// TIA Portal V18 export
// export: Created 2025-12-01T12:38:33.634491Z, ExportSetting None, DisplayName Totally Integrated Automation Portal, DisplayVersion V18 Update 5, DisplayName TIA Portal Openness, DisplayVersion V18 Update 5, DisplayName TIA Portal Teamcenter Gateway, DisplayVersion V18, DisplayName TIA Portal Version Control Interface, DisplayVersion V18, DisplayName STEP 7 Professional, DisplayVersion V18 Update 5, DisplayName STEP 7 Safety, DisplayVersion V18, DisplayName WinCC Professional, DisplayVersion V18 Update 5
FUNCTION "ST10Cyl_interface31-40" : Void   // FC1023, LAD
{ S7_Optimized_Access := 'FALSE' }
// stored: AutoNumber false, SetENOAutomatically false
   VAR_INPUT
      AlwaysON : Bool;
      E_stop : Bool;
   END_VAR
   VAR_TEMP
      tTest : Bool;
   END_VAR
BEGIN

REGION Network 1 (SCL): Cylinder 31-40 IO Interface (SCL)

   //Cylinder31 IO  J-magnetLiftingLiftingCylinder
   //Input
   "ST10Cylinder".Cy[31].In.WorkPositionSensor := "iJ-magnetLiftingLiftingCylinderInWP";
   "ST10Cylinder".Cy[31].In.HomePositionSensor := "iJ-magnetLiftingLiftingCylinderInHP";
   //Output
   "oJ-magnetLiftingLiftingCylinderToWP" := "ST10Cylinder".Cy[31].Out.GoWorkPosition;
   "oJ-magnetLiftingLiftingCylinderToHP" := "ST10Cylinder".Cy[31].Out.GoHomePosition;

   //Cylinder32 IO  J-magnetLiftingPalletLocationCylinder
   //Input
   "ST10Cylinder".Cy[32].In.WorkPositionSensor := "iJ-magnetLiftingPalletLocationCylinderInWP";
   "ST10Cylinder".Cy[32].In.HomePositionSensor := "iJ-magnetLiftingPalletLocationCylinderInHP";
   //Output
   "oJ-magnetLiftingPalletLocationCylinderToWP" := "ST10Cylinder".Cy[32].Out.GoWorkPosition;
   "oJ-magnetLiftingPalletLocationCylinderToHP" := "ST10Cylinder".Cy[32].Out.GoHomePosition;

   //Cylinder33 IO  J-magnetLoadingStopperCylinder1
   //Input
   "ST10Cylinder".Cy[33].In.WorkPositionSensor := "oJ-magnetLoadingStopperCylinder1_ToWP";
   "ST10Cylinder".Cy[33].In.HomePositionSensor := "oJ-magnetLoadingStopperCylinder1_ToHP";
   //Output
   "oJ-magnetLoadingStopperCylinder1_ToWP" := "ST10Cylinder".Cy[33].Out.GoWorkPosition;
   "oJ-magnetLoadingStopperCylinder1_ToHP" := "ST10Cylinder".Cy[33].Out.GoHomePosition;

   //Cylinder34 IO  J-magnetLoadingStopperCylinder2
   //Input
   "ST10Cylinder".Cy[34].In.WorkPositionSensor := "oJ-magnetLoadingStopperCylinder2_ToWP";
   "ST10Cylinder".Cy[34].In.HomePositionSensor := "oJ-magnetLoadingStopperCylinder2_ToHP";
   //Output
   "oJ-magnetLoadingStopperCylinder2_ToWP" := "ST10Cylinder".Cy[34].Out.GoWorkPosition;
   "oJ-magnetLoadingStopperCylinder2_ToHP" := "ST10Cylinder".Cy[34].Out.GoHomePosition;

   //Cylinder35 IO  J-magnetLoadingStopperCylinder3
   //Input
   "ST10Cylinder".Cy[35].In.WorkPositionSensor := "oJ-magnetLoadingStopperCylinder3_ToWP";
   "ST10Cylinder".Cy[35].In.HomePositionSensor := "oJ-magnetLoadingStopperCylinder3_ToHP";
   //Output
   "oJ-magnetLoadingStopperCylinder3_ToWP" := "ST10Cylinder".Cy[35].Out.GoWorkPosition;
   "oJ-magnetLoadingStopperCylinder3_ToHP" := "ST10Cylinder".Cy[35].Out.GoHomePosition;

   //Cylinder36 J-magnetLoadingStopperCylinder4
   //Input
   "ST10Cylinder".Cy[36].In.WorkPositionSensor := "oJ-magnetLoadingStopperCylinder4_ToWP";
   "ST10Cylinder".Cy[36].In.HomePositionSensor := "oJ-magnetLoadingStopperCylinder4_ToHP";
   //Output
   "oJ-magnetLoadingStopperCylinder4_ToWP" := "ST10Cylinder".Cy[36].Out.GoWorkPosition;
   "oJ-magnetLoadingStopperCylinder4_ToHP" := "ST10Cylinder".Cy[36].Out.GoHomePosition;

   //Cylinder37 J-magnetTakeStopperCylinder1
   //Input
   "ST10Cylinder".Cy[37].In.WorkPositionSensor := "oJ-magnetTakeStopperCylinder1_ToWP";
   "ST10Cylinder".Cy[37].In.HomePositionSensor := "oJ-magnetTakeStopperCylinder1_ToHP";
   //Output
   "oJ-magnetTakeStopperCylinder1_ToWP" := "ST10Cylinder".Cy[37].Out.GoWorkPosition;
   "oJ-magnetTakeStopperCylinder1_ToHP" := "ST10Cylinder".Cy[37].Out.GoHomePosition;

   //Cylinder38 J-magnetTakeStopperCylinder2
   //Input
   "ST10Cylinder".Cy[38].In.WorkPositionSensor := "oJ-magnetTakeStopperCylinder2_ToWP";
   "ST10Cylinder".Cy[38].In.HomePositionSensor := "oJ-magnetTakeStopperCylinder2_ToHP";
   //Output
   "oJ-magnetTakeStopperCylinder2_ToWP" := "ST10Cylinder".Cy[38].Out.GoWorkPosition;
   "oJ-magnetTakeStopperCylinder2_ToHP" := "ST10Cylinder".Cy[38].Out.GoHomePosition;

   //Cylinder39 J-magnetTakeStopperCylinder3
   //Input
   "ST10Cylinder".Cy[39].In.WorkPositionSensor := "oJ-magnetTakeStopperCylinder3_ToWP";
   "ST10Cylinder".Cy[39].In.HomePositionSensor := "oJ-magnetTakeStopperCylinder3_ToHP";
   //Output
   "oJ-magnetTakeStopperCylinder3_ToWP" := "ST10Cylinder".Cy[39].Out.GoWorkPosition;
   "oJ-magnetTakeStopperCylinder3_ToHP" := "ST10Cylinder".Cy[39].Out.GoHomePosition;

   (*
   //Cylinder40 J-magnetLoadingStopperCylinder4_2
   // //Input
   "ST10Cylinder".Cy[40].In.WorkPositionSensor := "oJ-magnetLoadingStopperCylinder4_2";
   "ST10Cylinder".Cy[40].In.HomePositionSensor := NOT "oJ-magnetLoadingStopperCylinder4_2";
   // //Output
   "oJ-magnetLoadingStopperCylinder4_2" := "ST10Cylinder".Cy[40].Out.GoWorkPosition;
   "Feeding washer  lift Cylinder ToHP" := "ST10Cylinder".Cy[40].Out.GoHomePosition;
   *)
END_REGION

REGION Network 2: CY31 interface J-magnetLiftingLiftingCylinder
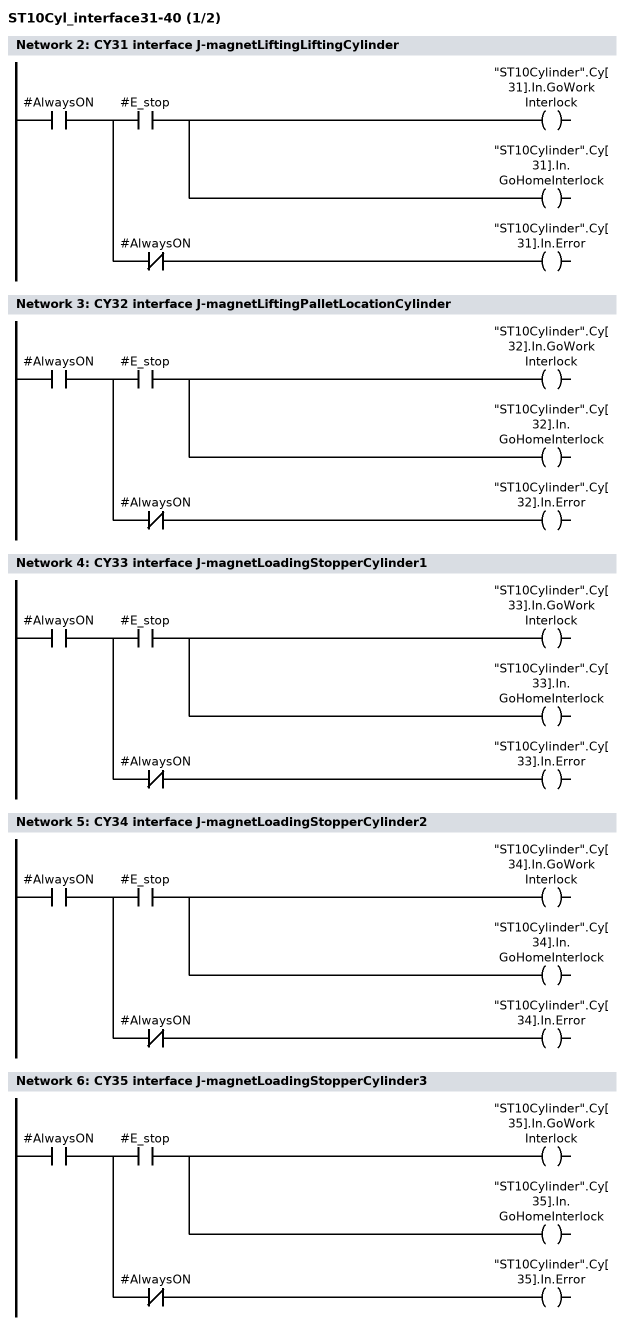
   RUNG wire#powerrail
      Contact( #AlwaysON )
      wire#w1
      Contact( #E_stop )
      wire#w2
      Coil( "ST10Cylinder".Cy[31].In.GoWorkInterlock )
   END_RUNG
   RUNG wire#w2
      Coil( "ST10Cylinder".Cy[31].In.GoHomeInterlock )
   END_RUNG
   RUNG wire#w1
      I_Contact( #AlwaysON )
      Coil( "ST10Cylinder".Cy[31].In.Error )
   END_RUNG
   // the same network as SCL:
   "ST10Cylinder".Cy[31].In.GoWorkInterlock := #AlwaysON AND #E_stop;
   "ST10Cylinder".Cy[31].In.GoHomeInterlock := #AlwaysON AND #E_stop;
   "ST10Cylinder".Cy[31].In.Error := #AlwaysON AND NOT #AlwaysON;
END_REGION

REGION Network 3: CY32 interface J-magnetLiftingPalletLocationCylinder
   RUNG wire#powerrail
      Contact( #AlwaysON )
      wire#w1
      Contact( #E_stop )
      wire#w2
      Coil( "ST10Cylinder".Cy[32].In.GoWorkInterlock )
   END_RUNG
   RUNG wire#w2
      Coil( "ST10Cylinder".Cy[32].In.GoHomeInterlock )
   END_RUNG
   RUNG wire#w1
      I_Contact( #AlwaysON )
      Coil( "ST10Cylinder".Cy[32].In.Error )
   END_RUNG
   // the same network as SCL:
   "ST10Cylinder".Cy[32].In.GoWorkInterlock := #AlwaysON AND #E_stop;
   "ST10Cylinder".Cy[32].In.GoHomeInterlock := #AlwaysON AND #E_stop;
   "ST10Cylinder".Cy[32].In.Error := #AlwaysON AND NOT #AlwaysON;
END_REGION

REGION Network 4: CY33 interface J-magnetLoadingStopperCylinder1
   RUNG wire#powerrail
      Contact( #AlwaysON )
      wire#w1
      Contact( #E_stop )
      wire#w2
      Coil( "ST10Cylinder".Cy[33].In.GoWorkInterlock )
   END_RUNG
   RUNG wire#w2
      Coil( "ST10Cylinder".Cy[33].In.GoHomeInterlock )
   END_RUNG
   RUNG wire#w1
      I_Contact( #AlwaysON )
      Coil( "ST10Cylinder".Cy[33].In.Error )
   END_RUNG
   // the same network as SCL:
   "ST10Cylinder".Cy[33].In.GoWorkInterlock := #AlwaysON AND #E_stop;
   "ST10Cylinder".Cy[33].In.GoHomeInterlock := #AlwaysON AND #E_stop;
   "ST10Cylinder".Cy[33].In.Error := #AlwaysON AND NOT #AlwaysON;
END_REGION

REGION Network 5: CY34 interface J-magnetLoadingStopperCylinder2
   RUNG wire#powerrail
      Contact( #AlwaysON )
      wire#w1
      Contact( #E_stop )
      wire#w2
      Coil( "ST10Cylinder".Cy[34].In.GoWorkInterlock )
   END_RUNG
   RUNG wire#w2
      Coil( "ST10Cylinder".Cy[34].In.GoHomeInterlock )
   END_RUNG
   RUNG wire#w1
      I_Contact( #AlwaysON )
      Coil( "ST10Cylinder".Cy[34].In.Error )
   END_RUNG
   // the same network as SCL:
   "ST10Cylinder".Cy[34].In.GoWorkInterlock := #AlwaysON AND #E_stop;
   "ST10Cylinder".Cy[34].In.GoHomeInterlock := #AlwaysON AND #E_stop;
   "ST10Cylinder".Cy[34].In.Error := #AlwaysON AND NOT #AlwaysON;
END_REGION

REGION Network 6: CY35 interface J-magnetLoadingStopperCylinder3
   RUNG wire#powerrail
      Contact( #AlwaysON )
      wire#w1
      Contact( #E_stop )
      wire#w2
      Coil( "ST10Cylinder".Cy[35].In.GoWorkInterlock )
   END_RUNG
   RUNG wire#w2
      Coil( "ST10Cylinder".Cy[35].In.GoHomeInterlock )
   END_RUNG
   RUNG wire#w1
      I_Contact( #AlwaysON )
      Coil( "ST10Cylinder".Cy[35].In.Error )
   END_RUNG
   // the same network as SCL:
   "ST10Cylinder".Cy[35].In.GoWorkInterlock := #AlwaysON AND #E_stop;
   "ST10Cylinder".Cy[35].In.GoHomeInterlock := #AlwaysON AND #E_stop;
   "ST10Cylinder".Cy[35].In.Error := #AlwaysON AND NOT #AlwaysON;
END_REGION

REGION Network 7: CY36 interface J-magnetLoadingStopperCylinder4
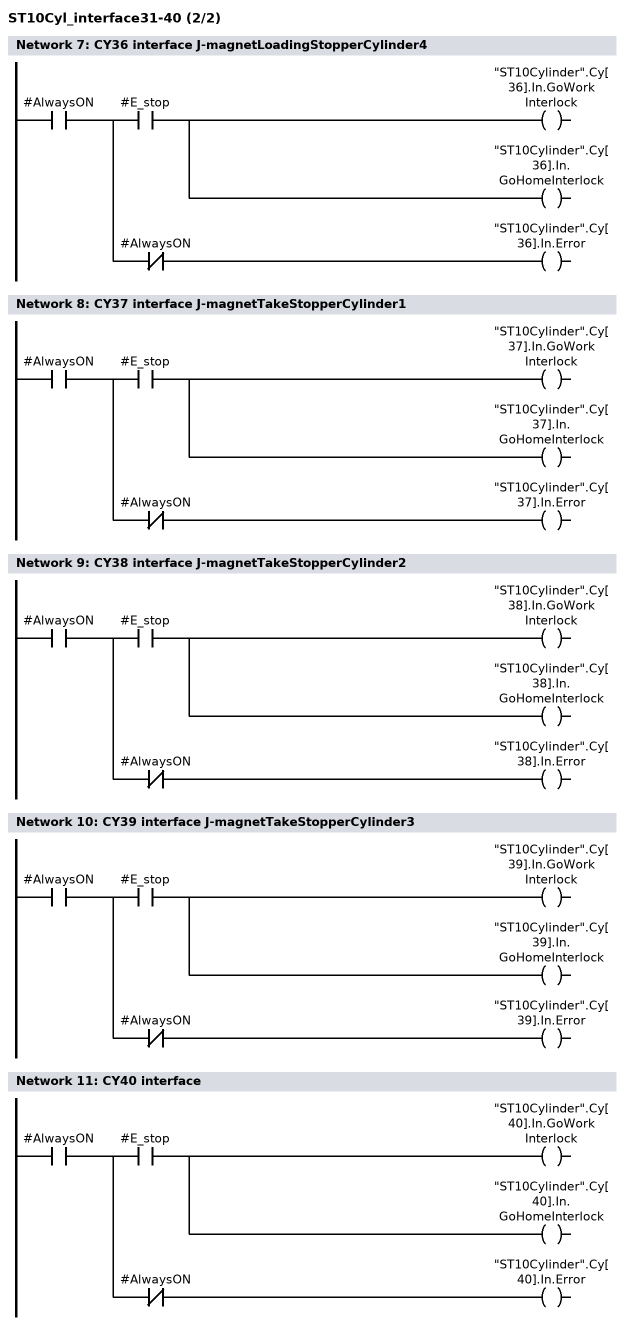
   RUNG wire#powerrail
      Contact( #AlwaysON )
      wire#w1
      Contact( #E_stop )
      wire#w2
      Coil( "ST10Cylinder".Cy[36].In.GoWorkInterlock )
   END_RUNG
   RUNG wire#w2
      Coil( "ST10Cylinder".Cy[36].In.GoHomeInterlock )
   END_RUNG
   RUNG wire#w1
      I_Contact( #AlwaysON )
      Coil( "ST10Cylinder".Cy[36].In.Error )
   END_RUNG
   // the same network as SCL:
   "ST10Cylinder".Cy[36].In.GoWorkInterlock := #AlwaysON AND #E_stop;
   "ST10Cylinder".Cy[36].In.GoHomeInterlock := #AlwaysON AND #E_stop;
   "ST10Cylinder".Cy[36].In.Error := #AlwaysON AND NOT #AlwaysON;
END_REGION

REGION Network 8: CY37 interface J-magnetTakeStopperCylinder1
   RUNG wire#powerrail
      Contact( #AlwaysON )
      wire#w1
      Contact( #E_stop )
      wire#w2
      Coil( "ST10Cylinder".Cy[37].In.GoWorkInterlock )
   END_RUNG
   RUNG wire#w2
      Coil( "ST10Cylinder".Cy[37].In.GoHomeInterlock )
   END_RUNG
   RUNG wire#w1
      I_Contact( #AlwaysON )
      Coil( "ST10Cylinder".Cy[37].In.Error )
   END_RUNG
   // the same network as SCL:
   "ST10Cylinder".Cy[37].In.GoWorkInterlock := #AlwaysON AND #E_stop;
   "ST10Cylinder".Cy[37].In.GoHomeInterlock := #AlwaysON AND #E_stop;
   "ST10Cylinder".Cy[37].In.Error := #AlwaysON AND NOT #AlwaysON;
END_REGION

REGION Network 9: CY38 interface J-magnetTakeStopperCylinder2
   RUNG wire#powerrail
      Contact( #AlwaysON )
      wire#w1
      Contact( #E_stop )
      wire#w2
      Coil( "ST10Cylinder".Cy[38].In.GoWorkInterlock )
   END_RUNG
   RUNG wire#w2
      Coil( "ST10Cylinder".Cy[38].In.GoHomeInterlock )
   END_RUNG
   RUNG wire#w1
      I_Contact( #AlwaysON )
      Coil( "ST10Cylinder".Cy[38].In.Error )
   END_RUNG
   // the same network as SCL:
   "ST10Cylinder".Cy[38].In.GoWorkInterlock := #AlwaysON AND #E_stop;
   "ST10Cylinder".Cy[38].In.GoHomeInterlock := #AlwaysON AND #E_stop;
   "ST10Cylinder".Cy[38].In.Error := #AlwaysON AND NOT #AlwaysON;
END_REGION

REGION Network 10: CY39 interface J-magnetTakeStopperCylinder3
   RUNG wire#powerrail
      Contact( #AlwaysON )
      wire#w1
      Contact( #E_stop )
      wire#w2
      Coil( "ST10Cylinder".Cy[39].In.GoWorkInterlock )
   END_RUNG
   RUNG wire#w2
      Coil( "ST10Cylinder".Cy[39].In.GoHomeInterlock )
   END_RUNG
   RUNG wire#w1
      I_Contact( #AlwaysON )
      Coil( "ST10Cylinder".Cy[39].In.Error )
   END_RUNG
   // the same network as SCL:
   "ST10Cylinder".Cy[39].In.GoWorkInterlock := #AlwaysON AND #E_stop;
   "ST10Cylinder".Cy[39].In.GoHomeInterlock := #AlwaysON AND #E_stop;
   "ST10Cylinder".Cy[39].In.Error := #AlwaysON AND NOT #AlwaysON;
END_REGION

REGION Network 11: CY40 interface
   RUNG wire#powerrail
      Contact( #AlwaysON )
      wire#w1
      Contact( #E_stop )
      wire#w2
      Coil( "ST10Cylinder".Cy[40].In.GoWorkInterlock )
   END_RUNG
   RUNG wire#w2
      Coil( "ST10Cylinder".Cy[40].In.GoHomeInterlock )
   END_RUNG
   RUNG wire#w1
      I_Contact( #AlwaysON )
      Coil( "ST10Cylinder".Cy[40].In.Error )
   END_RUNG
   // the same network as SCL:
   "ST10Cylinder".Cy[40].In.GoWorkInterlock := #AlwaysON AND #E_stop;
   "ST10Cylinder".Cy[40].In.GoHomeInterlock := #AlwaysON AND #E_stop;
   "ST10Cylinder".Cy[40].In.Error := #AlwaysON AND NOT #AlwaysON;
END_REGION
END_FUNCTION
